PROGRAM TEMP_MONITOR
VAR
		WaterCooling1: FB_WATERCOOLING;	
END_VAR

WaterCooling1(HEATER:=GVL.ox_HEATER,TEMP_SENSOR:=GVL.id_TEMP_SENSOR);

END_PROGRAM

(* stored: Version 1.1.0.1, ProductVersion 3.1.4024.15
   POU TEMP_MONITOR: Id {207a7309-f67d-4d97-8914-0c83f9d25e13}, SpecialFunc None *)
